//enum of states
{attribute 'strict'}
{attribute 'to_string'}
{attribute 'qualified_only'}
TYPE eTpc :
(
	//NOTE @ copy of this enum, adapt existing state names:
	Disabled := -1, //-1: to make sure the code for disabling fires
	TotalReset,
	Initialise,
	Rest
)INT;
END_TYPE

//info on attributes:
//strict 			: don't allow mixing of types
//to_string			: allows the enum to be converted to string
//qualified_only 	: forces the user to start witht the type name (to avoid the situation that accidentially another enum is used)

(* stored: Version 1.1.0.1
   DUT eTpc: Id {d3d3b2c1-1eef-4965-bd65-c52c8f932a0a} *)
